TYPE U_OdriveErrorBytes :
UNION
    stOdriveError : ST_OdriveError;
    aBytes : ARRAY[0..7] OF BYTE;
END_UNION
END_TYPE

(* stored: Version 1.1.0.1
   DUT U_OdriveErrorBytes: Id {4d090813-57c5-4fb8-b1be-4286f5823ecb} *)
